{attribute 'qualified_only'}
VAR_GLOBAL
	Reset_All:  BOOL;
	MQTT_Enable:  BOOL;
	OPC_Enable:  Bool;
END_VAR

(* stored: Version 1.1.0.1
   GVL System_Control_GVL: Id {67ec144b-997a-4ded-930e-76cdf75996df} *)
